{attribute 'linkalways'} 
{attribute 'no_explicit_call' := 'This FB is a CLASS and must be accessed using methods or properties'}
{attribute 'enable_dynamic_creation'}
FUNCTION_BLOCK Node_F_VN_ConnectedComponents EXTENDS VisionNode
VAR
    ipSrcImage : _ITcVnImage;
    ipLabelImage : _ITcVnImage;
    nLabels : _DINT(0);
    hrPrev : _HRESULT(S_OK);
	hresult : _HRESULT(S_OK);
END_VAR

METHOD PUBLIC  Clone : I_Node
VAR
	pNode : POINTER TO Node_F_VN_ConnectedComponents;
END_VAR
pNode := __NEW(Node_F_VN_ConnectedComponents);
Clone := pNode^;
END_METHOD

METHOD FB_init : BOOL
VAR_INPUT
	bInitRetains : BOOL; // if TRUE, the retain variables are initialized (warm start / cold start)
	bInCopyCode : BOOL;  // if TRUE, the instance afterwards gets moved into the copy code (online change)
END_VAR
AddInput('ipSrcImage', ipSrcImage);
AddInput('hrPrev', hrPrev);
AddOutput('ipLabelImage', ipLabelImage);
AddOutput('nLabels', nLabels);
AddOutput('hresult', hresult);
END_METHOD

METHOD PROTECTED OnExecute
hresult.Value := F_VN_ConnectedComponents(
	ipSrcImage := ipSrcImage.Value,
    ipLabelImage := ipLabelImage.Value,
    nLabels := nLabels.Value,
	hrPrev:= hrPrev.Value);
END_METHOD

METHOD PUBLIC PreExecutionCheck
VAR_INPUT
	Check : I_PreExecutionChecks;
END_VAR
Check.IsTrue(ipSrcImage.IsValid, 'ipSrcImage must contain an image');
Check.IsTrue(ipSrcImage.IsPixelDepth(8), 'ipSrcImage must be 8 bit pixel depth');
Check.IsTrue(ipSrcImage.HasChannelCount(1), 'ipSrcImage must contain 1 channel');
END_METHOD

END_FUNCTION_BLOCK

(* stored: Version 1.1.0.1, ProductVersion 3.1.4024.13
   POU Node_F_VN_ConnectedComponents: Id {f6f414bb-cbff-4683-a10f-e6fea201c87c}, SpecialFunc None
   Folder Constructor: Id {6c741be2-af38-4d28-b389-910042ed9624}
   Method Clone: Id {ee00e778-88d3-4192-805d-999294906de7}
   Method FB_init: Id {fb3d5590-15fb-4175-a1af-333cc01b03f9}
   Method OnExecute: Id {6b93925b-d431-48e2-81f1-165309357a90}
   Method PreExecutionCheck: Id {8877735e-cd02-4432-9d17-1da88dd6fb1f} *)
